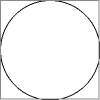
VISUALIZATION Visualization  // 100x100
    Ellipse (0,0 100x100)
        p3560616238: MAIN.iRBig - 50
        p1097714728: ((MAIN.iRBig) / 50 ) * 1000
        p2738717112: MAIN.iRBig - 50
    Ellipse (0,0 100x100)
        p3560616238: MAIN.iRSmall - 50 + MAIN.rSmallX
        p1097714728: ((MAIN.iRSmall) / 50 ) * 1000
        p2738717112: MAIN.iRSmall - 50 + MAIN.rSmallY
END_VISUALIZATION

(* stored: Version 1.1.0.1
   Visu Visualization: Id {f406055f-0ee7-4e29-8887-32c010c4638f} *)
